{attribute 'qualified_only'}
VAR_GLOBAL
    // InValues
    {attribute 'OPC.UA.DA' := '1'}
    {attribute 'OPC.UA.DA.StructuredType' := '1'}
    g_stBigBagMassStoreInValues   : ST_BigBagActualMassStoreInValues;


    // Status
    {attribute 'OPC.UA.DA' := '1'}
    {attribute 'OPC.UA.DA.StructuredType' := '1'}
    g_stBigBagMassStoreStatus     : ST_BigBagActualMassStoreStatus;
	
	// OutValues
    {attribute 'OPC.UA.DA' := '1'}
    {attribute 'OPC.UA.DA.StructuredType' := '1'}
    g_stBigBagMassStoreOutValues   : ST_BigBagActualMassStoreOutValues;
END_VAR

(* stored: Version 1.1.0.1, ProductVersion 3.1.4024.16
   GVL GVL_BigBagActualMassStore: Id {33575c06-1249-4a64-bf35-c2c31a820186} *)
